(* IEC 61131-3 sources: volt/packages/volt-lsp-iec/test-corpus/lenze-mid/Device/Plc Logic/Application/A55_VarLists, 21 files *)

(* ---- Bugs.gvl ---- *)
{attribute 'qualified_only'}
{attribute 'symbol' := 'readwrite'}
VAR_GLOBAL
	checkconnection: BOOL;
	reportConnectionAlive:BOOL;
	restart: BOOL;
END_VAR

(* ---- CTE.gvl ---- *)
{attribute 'qualified_only'}
VAR_GLOBAL CONSTANT
	//TODO
	posCigarPresentOutfeed	: INT:=88;
	ct_ArraySizeCheckRegister : INT:=150;

END_VAR

(* ---- Data_Exchange_Motion.gvl ---- *)
{attribute 'qualified_only'}
VAR_GLOBAL
Servo_VirtualMaster: sUDT_VirtualMasterComm_Drive;

Servo_MainDrive: sUDT_ServoComm_Drive;
Servo_WrappingDevice: sUDT_ServoComm_Drive;
Servo_SideCorrection: sUDT_ServoComm_Drive;

FQI_FeedforwardADS : sUDT_FQIComm_Drive;
FQI_FeedforwardATF : sUDT_FQIComm_Drive;
FQI_ElevatorATF : sUDT_FQIComm_Drive;
FQI_Fan : sUDT_FQIComm_Drive;
FQI_Bobbin : sUDT_FQIComm_Drive;
BobbinTorque: DINT;

FeedForwardWrapper : sUDT_BasicMovementComm_Drive ;
END_VAR

(* ---- db_CheckRegister.gvl ---- *)
{attribute 'qualified_only'}
{attribute 'symbol' := 'readwrite'}
VAR_GLOBAL
	//Positie		: ARRAY[0..CTE.ct_ArraySizeCheckRegister] OF cUDT_ShiftRegister_Positie;
	Positie		: ARRAY[0..CTE.ct_ArraySizeCheckRegister] OF cUDT_ShiftRegister_Positie;
	EmptyCheckRegister : cUDT_ShiftRegister_Positie;
	CheckRegisterError	: BOOL;
END_VAR

(* ---- DB_Kantcorrectie.gvl ---- *)
{attribute 'qualified_only'}
{attribute 'symbol' := 'readwrite'}
VAR_GLOBAL PERSISTENT
	CopyMeasuredToLight: BOOL;
	CopyMeasuredToDark: BOOL;
	MeasuredValue		: INT;
	MeasuredValueReal	: REAL;
	Percentage			: REAL;
	Percentage10		: INT ;
	Setpoint			: INT;
	CopiedValueReal		: REAL;
	CopiedValueInt		: INT;
	LightValue			: INT:=100;
	DarkValue			: INT:=5;
	NoWrapperValue		: INT;
	DeviationNoWrapper	: INT;
	NoWrapperPercentage	: INT;
	SpareInt_2			: INT;

END_VAR

(* ---- db_MeanValuesSideCorrectionSensor.gvl ---- *)
{attribute 'qualified_only'}
VAR_GLOBAL PERSISTENT
	MeasurementValues	: ARRAY[0..50] OF INT ;
END_VAR

(* ---- Droger_Data.gvl ---- *)
{attribute 'qualified_only'}
VAR_GLOBAL
	Cor_denumerator: INT:=1;
	Cor_numerator: INT:=1;
	Act_sync_pos: INT:=1;
	Set_sync_pos: INT:=1;
END_VAR

(* ---- HMI_Interface.gvl ---- *)
{attribute 'qualified_only'}
VAR_GLOBAL
	ScreenNumber 	: sUDT_HMI_Interface_ScreenNumber;
END_VAR

(* ---- HMI_Var.gvl ---- *)
{attribute 'qualified_only'}
{attribute 'symbol' := 'readwrite'}
VAR_GLOBAL PERSISTENT RETAIN
SpareRecipe : ARRAY[0..19] OF BYTE;
RecipeNumber : Int;
DataRecordNumber : Int;
DataRecordName : String;
DownloadStatus : Int;
ResetAlarmLogging : Bool;
ForceOutputs : Bool;
RE_ForceOutputs : Bool;
Test_Prod : Bool;
Btn_Spraying : Bool;
Btn_BunchSupply : Bool;
Btn_StopLeafCarrier : Bool;
ReleaseBrake : Bool;
ManControl_1 : Bool;
ManControl_2 : Bool;
ManControl_3 : Bool;
TrayfillerActive : Bool;
Btn_DryerOn : Bool;
Btn_Cleaning : Bool;
Btn_SetIP : Bool;
HMI_AHWF_fast_winding : Bool;
SpareBool21_7 : Bool;
Led_K_Buttons : Word;
Password : Int;
HMI_AHWF_positioningType : Bool;
HMI_AHWF_StartPos : Bool;
CMD_DateTime : Bool;
Mach1: sUDT_HMIVar_Mach1;

END_VAR

(* ---- LST_General.gvl ---- *)
//{attribute 'qualified_only'}
VAR_GLOBAL
	AlwaysOn							: BOOL :=1;
	AlwaysOff							: BOOL :=0;
	FirstCycle							: BOOL:=1;

	FF50ms								: BOOL;
	Imp100ms							: BOOL;

	FF100ms								: BOOL;
	Imp200ms							: BOOL;

	FF500ms								: BOOL;
	Imp1s								: BOOL;

	FF1s								: BOOL;

	StartUpDelayPLC						: BOOL;

END_VAR

(* ---- LST_InputsOutputs.gvl ---- *)
{attribute 'qualified_only'}
VAR_GLOBAL

	//inputs
I100_0_AirpressureOK : BOOL;
I100_1_Pushbutton_start_OP0a : BOOL;
I100_2_Pushbutton_stop_OP0a : BOOL;
I100_3_Selector_switch_auto_manual_OP0a : BOOL;
I100_4_Pushbutton_request_glue_OP0a : BOOL;
I100_5_ConfigSelectionRightMachine : BOOL;
I100_6_Greasing_system_empty : BOOL;
I100_7_Spare : BOOL;

I101_0_Wrapper_present : BOOL;
I101_1_FC_Bunch_present : BOOL;
I101_2_Cigar_present : BOOL;
I101_3_Water_level_control : BOOL;
I101_4_Level_bunch_magazine : BOOL;
I101_5_Spare : BOOL;
I101_6_Toggle_greasing_cycle : BOOL;
I101_7_Spare : BOOL;

I132_0_Thermal_guards_OK : BOOL;
I132_1_PB_Start_OP2a : BOOL;
I132_2_PB_Stop_OP2a : BOOL;
I132_3_SW_Auto_Man : BOOL;
I132_4_Spare : BOOL;
I132_5_Spare : BOOL;
I132_6_Tray_down : BOOL;
I132_7_Tray_up : BOOL;

I133_0_PROX_Dryer_closed : BOOL;
I133_1_PROX_zero_position_transport_ADS : BOOL;
I133_2_Cigar_detected_at_cross_over : BOOL;
I133_3_PROX_zero_position_transport_ATF : BOOL;
I133_4_Cigar_detected_at_inpusher : BOOL;
I133_5_Spare : BOOL;
I133_6_PROX_inpusher_retracted : BOOL;
I133_7_PROX_inpusher_at_tray : BOOL;

I136_0_PROX_Elevator_above : BOOL;
I136_1_PROX_Elevator_below : BOOL;
I136_2_PROX_pulse_counter_elevator : BOOL;
I136_3_FC_Position_tray_OK : BOOL;
I136_4_PROX_Infeed_conveyor_initial_position : BOOL;
I136_5_PROX_Infeed_conveyor_at_elevator : BOOL;
I136_6_FC_Guard_tray_from_elevator : BOOL;
I136_7_FC_Outfeed_conveyor_full : BOOL;

I137_0_Spare : BOOL;
I137_1_Spare : BOOL;
I137_2_Spare : BOOL;
I137_3_Spare : BOOL;
I137_4_Spare : BOOL;
I137_5_Spare : BOOL;
I137_6_Spare : BOOL;
I137_7_Spare : BOOL;

Q100_0_Pilot_light_Alarm_green_ : BOOL;
Q100_1_Pilot_light_Alarm_orange_ : BOOL;
Q100_2_Pilot_light_Alarm_red_ : BOOL;
Q100_3_Pilot_light_Alarm_buzzer_ : BOOL;
Q100_4_Spare : BOOL;
Q100_5_Signal_lamp_Start : BOOL;
Q100_6_Signal_lamp_Stop : BOOL;
Q100_7_Activate_greasing_system : BOOL;

Q101_0_REL_release_brake : BOOL;
Q101_1_PNV_Waterlevel_control : BOOL;
Q101_2_Enable_GluePump : BOOL;
Q101_3_Spare : BOOL;
Q101_4_Spare : BOOL;
Q101_5_Spare : BOOL;
Q101_6_Spare : BOOL;
Q101_7_Spare : BOOL;

Q132_0_SL_Start_OP2a : BOOL;
Q132_1_SL_Stop_OP2a : BOOL;
Q132_2_Enable_power_controllers : BOOL;
Q132_3_Spare : BOOL;
Q132_4_CT_Fan_dryer : BOOL;
Q132_5_Spare : BOOL;
Q132_6_PNV_Inpusher : BOOL;
Q132_7_PNV_tilting_inpusher : BOOL;

Q133_0_Spare : BOOL;
Q133_1_Spare : BOOL;
Q133_2_Spare : BOOL;
Q133_3_Spare : BOOL;
Q133_4_Spare : BOOL;
Q133_5_InfeedConv_Fwd : BOOL;
Q133_6_InfeedConv_Rev : BOOL;
Q133_7_OutfeedConv_Fwd : BOOL;

Q136_0_Spare : BOOL;
Q136_1_Spare : BOOL;
Q136_2_Spare : BOOL;
Q136_3_Spare : BOOL;
Q136_4_Spare : BOOL;
Q136_5_Spare : BOOL;
Q136_6_Spare : BOOL;
Q136_7_Spare : BOOL;

Q137_0_Spare : BOOL;
Q137_1_Spare : BOOL;
Q137_2_Spare : BOOL;
Q137_3_Spare : BOOL;
Q137_4_Spare : BOOL;
Q137_5_Spare : BOOL;
Q137_6_Spare : BOOL;
Q137_7_Spare : BOOL;

{attribute 'symbol' := 'readwrite'}
IW340_LeafCoverageSensor			: INT;
{attribute 'symbol' := 'readwrite'}
Serv_QW320 : BOOL;
{attribute 'symbol' := 'readwrite'}
Serv_QW322 : BOOL;
{attribute 'symbol' := 'readwrite'}
Serv_QW324 : BOOL;

{attribute 'symbol' := 'readwrite'}
Serv_IB100 : BYTE;
{attribute 'symbol' := 'readwrite'}
Serv_IB101 : BYTE;
{attribute 'symbol' := 'readwrite'}
Serv_IB132 : BYTE;
{attribute 'symbol' := 'readwrite'}
Serv_IB133 : BYTE;
{attribute 'symbol' := 'readwrite'}
Serv_IB136 : BYTE;
{attribute 'symbol' := 'readwrite'}
Serv_IB137 : BYTE;
{attribute 'symbol' := 'readwrite'}
Serv_QB100 : BYTE;
{attribute 'symbol' := 'readwrite'}
Serv_QB101 : BYTE;
{attribute 'symbol' := 'readwrite'}
Serv_QB132 : BYTE;
{attribute 'symbol' := 'readwrite'}
Serv_QB133 : BYTE;
{attribute 'symbol' := 'readwrite'}
Serv_QB136 : BYTE;
{attribute 'symbol' := 'readwrite'}
Serv_QB137 : BYTE;
{attribute 'symbol' := 'readwrite'}
IW342_Spare : BOOL;
IW344_Spare : BOOL;
IW346_Spare : BOOL;

{attribute 'symbol' := 'readwrite'}
SMC_B0: BYTE;
{attribute 'symbol' := 'readwrite'}
SMC_B1: BYTE;
{attribute 'symbol' := 'readwrite'}
SMC_B2: BYTE;
{attribute 'symbol' := 'readwrite'}
SMC_B3: BYTE;

END_VAR

(* ---- Mach1.gvl ---- *)
{attribute 'qualified_only'}
{attribute 'symbol' := 'readwrite'}
VAR_GLOBAL
	Genflags				: UDT_GeneralFlags;
END_VAR

(* ---- Mach1_Alarms.gvl ---- *)
{attribute 'symbol' := 'readwrite'}
VAR_GLOBAL
	Mach1_Alarms	: scAlarmsDB;
	dwErrorWord1	: DWORD;
	dwErrorWord2	: DWORD;
	dwErrorWord3	: DWORD;
	dwErrorWord4	: DWORD;
END_VAR

(* ---- Mach1_AuxData.gvl ---- *)
{attribute 'qualified_only'}
VAR_GLOBAL
	AllDriveReferencingDone : BOOL;
SetDrivesInSync : Bool;
SetDrivesInLock : Bool;
AllDrivesInLock : Bool;
StartpulseDryer : Bool;
SetBuzzer : Bool;
MemContinuousGluePumping : Bool;
MemStopLeafCarrier : Bool;
MemStopCleaning : Bool;
DelayAfterDoorsActuallyClosed : Bool;
PhotocellBunchHasBeenOff : BOOL;
PhotocellCigarHasBeenOff : BOOL;
ScreenForOperatorSettingsActivated : Bool;
GlueWeighingCycleStarted : Bool;
NumberOfMutingCyclesReached : Bool;
MemLowerSpeedBecauseOfNoWrapper : Bool;
MemWrapperPresentForLeafCarrier : Bool;
MemWrapperPassedUnderTheSensor : Bool;
MemWrapperDetected_ResetLimitedSpeed : Bool;
BlockBunchInfeed : Bool;
MainDriveHomed : Bool;
RollingDeviceHomed : Bool;
DTA_Homed : Bool;
AllDrivesHomed : Bool;
CurrentCycleHasOutfeedError : Bool;
PreviousCycleHasOutfeedError : Bool;
MemCigarAtCrossOver : Bool;
ADS_StopOnZeroPulse : BOOL;
{attribute 'symbol' := 'readwrite'}
TorqueCalibrationValue : DInt;
TrayfillerActive : BOOL;
CounterHighSpeedATF_ADS: INT;
{attribute 'symbol' := 'readwrite'}
MIDS_Active : BOOL;
{attribute 'symbol' := 'readwrite'}
VelWrapperTransp : DINT;
{attribute 'symbol' := 'readwrite'}
EnableGlueSprayCalibration: BOOL:=FALSE;

{attribute 'symbol' := 'readwrite'}
EnableManualHomeSetting: BOOL:=FALSE;

IEC_TIMERS: cUDT_MachAuxData_Timers;
Edge: cUDT_MachAuxData_Edge;
COUNTERS: cUDT_MachAuxData_Counters;
ShiftRegister: cUDT_MachAuxData_Shiftregister;
CamControls : cUDT_MachAuxData_CamControls;

END_VAR

(* ---- Mach1_Data.gvl ---- *)
{attribute 'qualified_only'}
{attribute 'symbol' := 'readwrite'}
VAR_GLOBAL PERSISTENT RETAIN
MachineName : STRING;

AutoSpeed					: INT:=20;
ManualSpeed					: INT:=10;
CamControls					: cUDT_MachData_CamControls;
Timers						: cUDT_MachData_Timers;
Drives						: cUDT_MachData_Drives;
Counters					: cUDT_MachData_Counters;
Settings					: cUDT_MachData_Settings;
Dryer						: cUDT_MachData_Dryer;
TrayFiller					: cUDT_MachData_Trayfiller;

END_VAR

(* ---- Mach1_Safety.gvl ---- *)
{attribute 'qualified_only'}
{attribute 'symbol' := 'readwrite'}
VAR_GLOBAL
	Control	:	udtSafety_Control;
	Status :	udtSafety_Status;
END_VAR

(* ---- PersistentVars.gvl ---- *)
{attribute 'qualified_only'}
VAR_GLOBAL PERSISTENT RETAIN
// Generated instance path of persistent variable
	Mach1_MIDS.Mach1_Drives_DB.ServoMainDrive.STATE_Prehoming: BOOL;
	// Generated instance path of persistent variable
	Mach1_MIDS.Mach1_Drives_DB.ServoWrappingDevice.STATE_Prehoming: BOOL;
	// Generated instance path of persistent variable
	Mach1_MIDS.Mach1_Drives_DB.ServoSideCorrection.STATE_Prehoming: BOOL;
	// Generated instance path of persistent variable
	Mach1_MIDS.Mach1_Drives_DB.ServoMainDrive.STATE_HomePosNOK: BOOL;
	// Generated instance path of persistent variable
	Mach1_MIDS.Mach1_Drives_DB.ServoWrappingDevice.STATE_HomePosNOK: BOOL;
	// Generated instance path of persistent variable
	Mach1_MIDS.Mach1_Drives_DB.ServoSideCorrection.STATE_HomePosNOK: BOOL;
	// Generated instance path of persistent variable
	Mach1_MIDS.Mach1_Drives_DB.ServoMainDrive.STATE_HomePOSOK: BOOL;
	// Generated instance path of persistent variable
	Mach1_MIDS.Mach1_Drives_DB.ServoWrappingDevice.STATE_HomePOSOK: BOOL;
	// Generated instance path of persistent variable
	Mach1_MIDS.Mach1_Drives_DB.ServoSideCorrection.STATE_HomePOSOK: BOOL;
	// Generated instance path of persistent variable
	Mach1_MIDS.Mach1_Drives_DB.ServoMainDrive.STATE_WaitingForEnable: BOOL;
	// Generated instance path of persistent variable
	Mach1_MIDS.Mach1_Drives_DB.ServoWrappingDevice.STATE_WaitingForEnable: BOOL;
	// Generated instance path of persistent variable
	Mach1_MIDS.Mach1_Drives_DB.ServoSideCorrection.STATE_WaitingForEnable: BOOL;
	// Generated instance path of persistent variable
	Mach1_MIDS.Mach1_Drives_DB.ServoMainDrive.STATE_Synchronising: BOOL;
	// Generated instance path of persistent variable
	Mach1_MIDS.Mach1_Drives_DB.ServoWrappingDevice.STATE_Synchronising: BOOL;
	// Generated instance path of persistent variable
	Mach1_MIDS.Mach1_Drives_DB.ServoSideCorrection.STATE_Synchronising: BOOL;
	// Generated instance path of persistent variable

	// Generated instance path of persistent variable
	Mach1_MIDS.IDB_Dryer.stReFeedForward: R_TRIG;
	// Generated instance path of persistent variable
	Mach1_MIDS.IDB_Dryer.TMR_IntervalTimerEmptying: TON;
	// Generated instance path of persistent variable
	Mach1_MIDS.IDB_Dryer.stFaultDryerOpened: sr;
	// Generated instance path of persistent variable
	Mach1_MIDS.IDB_Dryer.stReStopFeedForward: R_TRIG;
	// Generated instance path of persistent variable
	Mach1_MIDS.IDB_Dryer.TMR_HeaterTimeOut: TON;
	// Generated instance path of persistent variable
	AHWF.IDB_WSM.stRestposition: BOOL;
	// Generated instance path of persistent variable
	AHWF.IDB_WSM.stSupplyWrapper: BOOL;
	// Generated instance path of persistent variable
	AHWF.IDB_WSM.stWrapperPresent: BOOL;
	// Generated instance path of persistent variable
	AHWF.IDB_WSM.stNoWrapper: BOOL;
	// Generated instance path of persistent variable
	AHWF.IDB_WSM.stPhotocellWrapperFault: BOOL;
	// Generated instance path of persistent variable
	AHWF.IDB_WSM.stFeedForward: BOOL;
	// Generated instance path of persistent variable
	Mach1_Data.AutoSpeed: INT;
	// Generated instance path of persistent variable
	Mach1_Data.ManualSpeed: INT;
	// Generated instance path of persistent variable
	Mach1_Data.CamControls: cUDT_MachData_CamControls;
	// Generated instance path of persistent variable
	Mach1_Data.Timers: cUDT_MachData_Timers;
	// Generated instance path of persistent variable
	Mach1_Data.Drives: cUDT_MachData_Drives;
	// Generated instance path of persistent variable
	Mach1_Data.Counters: cUDT_MachData_Counters;
	// Generated instance path of persistent variable
	Mach1_Data.Settings: cUDT_MachData_Settings;
	// Generated instance path of persistent variable
	Mach1_Data.Dryer: cUDT_MachData_Dryer;
	// Generated instance path of persistent variable
	Mach1_Data.TrayFiller: cUDT_MachData_Trayfiller;
	// Generated instance path of persistent variable
	db_MeanValuesSideCorrectionSensor.MeasurementValues: ARRAY [0..50] OF INT;
	// Generated instance path of persistent variable
	DB_Kantcorrectie.MeasuredValue: INT;
	// Generated instance path of persistent variable
	DB_Kantcorrectie.MeasuredValueReal: REAL;
	// Generated instance path of persistent variable
	DB_Kantcorrectie.Percentage: REAL;
	// Generated instance path of persistent variable
	DB_Kantcorrectie.Percentage10: INT;
	// Generated instance path of persistent variable
	DB_Kantcorrectie.Setpoint: INT;
	// Generated instance path of persistent variable
	DB_Kantcorrectie.CopiedValueReal: REAL;
	// Generated instance path of persistent variable
	DB_Kantcorrectie.CopiedValueInt: INT;
	// Generated instance path of persistent variable
	DB_Kantcorrectie.LightValue: INT;
	// Generated instance path of persistent variable
	DB_Kantcorrectie.DarkValue: INT;
	// Generated instance path of persistent variable
	DB_Kantcorrectie.NoWrapperValue: INT;
	// Generated instance path of persistent variable
	DB_Kantcorrectie.DeviationNoWrapper: INT;
	// Generated instance path of persistent variable
	DB_Kantcorrectie.NoWrapperPercentage: INT;
	// Generated instance path of persistent variable
	DB_Kantcorrectie.SpareInt_2: INT;

	//manual added values
	//AxisPosMaindrive: SMC3_PersistPosition_Data;
	//AxisPosSidecorrection: SMC3_PersistPosition_Data;
	//AxisPosWrapper: SMC3_PersistPosition_Data;

	// Generated instance path of persistent variable
	Mach1_Data.MachineName: STRING;
	// Generated instance path of persistent variable
	Mach1_MotionControl.VirtualMaster_0.lrRetainPosition: LREAL;
	// Generated instance path of persistent variable
	DB_Kantcorrectie.CopyMeasuredToLight: BOOL;
	// Generated instance path of persistent variable
	DB_Kantcorrectie.CopyMeasuredToDark: BOOL;
	// Generated instance path of persistent variable
	HMI_Var.SpareRecipe: ARRAY [0..19] OF BYTE;
	// Generated instance path of persistent variable
	HMI_Var.RecipeNumber: INT;
	// Generated instance path of persistent variable
	HMI_Var.DataRecordNumber: INT;
	// Generated instance path of persistent variable
	HMI_Var.DataRecordName: STRING;
	// Generated instance path of persistent variable
	HMI_Var.DownloadStatus: INT;
	// Generated instance path of persistent variable
	HMI_Var.ResetAlarmLogging: BOOL;
	// Generated instance path of persistent variable
	HMI_Var.ForceOutputs: BOOL;
	// Generated instance path of persistent variable
	HMI_Var.RE_ForceOutputs: BOOL;
	// Generated instance path of persistent variable
	HMI_Var.Test_Prod: BOOL;
	// Generated instance path of persistent variable
	HMI_Var.Btn_Spraying: BOOL;
	// Generated instance path of persistent variable
	HMI_Var.Btn_BunchSupply: BOOL;
	// Generated instance path of persistent variable
	HMI_Var.Btn_StopLeafCarrier: BOOL;
	// Generated instance path of persistent variable
	HMI_Var.ReleaseBrake: BOOL;
	// Generated instance path of persistent variable
	HMI_Var.ManControl_1: BOOL;
	// Generated instance path of persistent variable
	HMI_Var.ManControl_2: BOOL;
	// Generated instance path of persistent variable
	HMI_Var.ManControl_3: BOOL;
	// Generated instance path of persistent variable
	HMI_Var.TrayfillerActive: BOOL;
	// Generated instance path of persistent variable
	HMI_Var.Btn_DryerOn: BOOL;
	// Generated instance path of persistent variable
	HMI_Var.Btn_Cleaning: BOOL;
	// Generated instance path of persistent variable
	HMI_Var.Btn_SetIP: BOOL;
	// Generated instance path of persistent variable
	HMI_Var.HMI_AHWF_fast_winding: BOOL;
	// Generated instance path of persistent variable
	HMI_Var.SpareBool21_7: BOOL;
	// Generated instance path of persistent variable
	HMI_Var.Led_K_Buttons: WORD;
	// Generated instance path of persistent variable
	HMI_Var.Password: INT;
	// Generated instance path of persistent variable
	HMI_Var.HMI_AHWF_positioningType: BOOL;
	// Generated instance path of persistent variable
	HMI_Var.HMI_AHWF_StartPos: BOOL;
	// Generated instance path of persistent variable
	HMI_Var.CMD_DateTime: BOOL;
	// Generated instance path of persistent variable
	HMI_Var.Mach1: sUDT_HMIVar_Mach1;
	// Generated instance path of persistent variable
	VersionInfo_DB.PLC_version: STRING := 'ghjhggj';
	// Generated instance path of persistent variable
	VersionInfo_DB.PLC_Version_Date: STRING := 'ghjhggj';
	// Generated instance path of persistent variable
	MM_PD.scDowntime: L_OEEA_Lib.scDowntime;
	// Generated instance path of persistent variable
	MM_PD.scPDinternal: L_OEEA_Lib.scInternalVar;
	// Generated instance path of persistent variable
	MM_PD.scPDinternalDowntime: L_OEEA_Lib.scInternalDownVar;
	// Generated instance path of persistent variable
	MM_PD.scPDProductionData: L_OEEA_Lib.scInternalProductionData;
	// Generated instance path of persistent variable
	MM_PD.scPDShiftDayIndex: L_OEEA_Lib.scPDShiftData;
	// Generated instance path of persistent variable
	MM_PD.scShiftHistory: L_OEEA_Lib.scVisuShiftHistory_base;
	// Generated instance path of persistent variable
	MM_PD.scShiftDowntimeHistory: ARRAY [1..3] OF L_OEEA_Lib.scDowntime_base;
	// Generated instance path of persistent variable
	MM_PD.scOEE_VisuPD: L_OEEA_Lib.scOEE_VisuPD := STRUCT(ascVisu_OUT_ShiftTargets := [STRUCT(rOEETarget := 90.0, rOEELowerLimit := 75.0, rOEECrucial := 65.0), STRUCT(rOEETarget := 90.0, rOEELowerLimit := 75.0, rOEECrucial := 65.0), STRUCT(rOEETarget := 90.0, rOEELowerLimit := 75.0, rOEECrucial := 65.0)]);
	// Generated instance path of persistent variable
	MM_PD.scSelectedProductRecipeHMI: L_OEEA_Lib.scProduct_base;
	// Generated instance path of persistent variable
	MM_PD.sActiveProductRecipe: STRING;
	// Generated instance path of persistent variable
	MM_PD.scActiveProductRecipe: L_OEEA_Lib.scProduct_base := STRUCT(rTechnicalCycleTime := REAL#1.5, rProductTarget := 15480.0, diTypeID := DINT#1, sTypeName := 'Sigar', iUnitProductID := INT#1, sUnitProduct := 'Sigars', iUnitSpeedID := INT#1, sUnitSpeed := 'Sigars/min.', rChangeOverTime := 60.0);
	// Generated instance path of persistent variable
	MM_PD.ascDaySchedules: ARRAY [1..L_OEEA_lib.uiDaySchedule] OF L_OEEA_Lib.scDaySchedule := [7(STRUCT(iNumberofShifts := UINT_TO_INT(L_OEEA_Lib.uiNoOfShifts), iNumberofBreaks := UINT_TO_INT(L_OEEA_lib.uiNoOfBreaks), ascShiftSchedule := [STRUCT(sShiftName := 'Morning', uiStartHour := UINT#6, uiStartMinute := UINT#30, uiEndHour := UINT#14, uiEndMinute := UINT#30, uiShiftNo := UINT#1, xActive := TRUE), STRUCT(sShiftName := 'Afternoon', uiStartHour := UINT#14, uiStartMinute := UINT#30, uiEndHour := UINT#22, uiEndMinute := UINT#30, uiShiftNo := UINT#2, xActive := TRUE), STRUCT(sShiftName := 'Night', uiStartHour := UINT#22, uiStartMinute := UINT#30, uiEndHour := UINT#6, uiEndMinute := UINT#30, uiShiftNo := UINT#3, xActive := TRUE)], ascSBreakSchedule := [STRUCT(sBreakName := 'Breakfast', uiStartHour := UINT#9, uiStartMinute := UINT#0, uiEndHour := UINT#9, uiEndMinute := UINT#10, uiShiftNo := UINT#1, xActive := TRUE), STRUCT(sBreakName := 'Lunch', uiStartHour := UINT#11, uiStartMinute := UINT#0, uiEndHour := UINT#11, uiEndMinute := UINT#30, uiShiftNo := UINT#1, xActive := TRUE), STRUCT(sBreakName := 'Tea Break', uiStartHour := UINT#13, uiStartMinute := UINT#0, uiEndHour := UINT#13, uiEndMinute := UINT#10, uiShiftNo := UINT#1, xActive := TRUE), STRUCT(sBreakName := 'Tea Break 1', uiStartHour := UINT#16, uiStartMinute := UINT#0, uiEndHour := UINT#16, uiEndMinute := UINT#10, uiShiftNo := UINT#2, xActive := TRUE), STRUCT(sBreakName := 'Dinner', uiStartHour := UINT#18, uiStartMinute := UINT#45, uiEndHour := UINT#19, uiEndMinute := UINT#15, uiShiftNo := UINT#2, xActive := TRUE), STRUCT(sBreakName := 'Tea Break 2', uiStartHour := UINT#20, uiStartMinute := UINT#45, uiEndHour := UINT#20, uiEndMinute := UINT#55, uiShiftNo := UINT#2, xActive := TRUE), STRUCT(sBreakName := 'Tea Break 1', uiStartHour := UINT#23, uiStartMinute := UINT#30, uiEndHour := UINT#23, uiEndMinute := UINT#40, uiShiftNo := UINT#3, xActive := TRUE), STRUCT(sBreakName := 'Dinner', uiStartHour := UINT#1, uiStartMinute := UINT#45, uiEndHour := UINT#2, uiEndMinute := UINT#12, uiShiftNo := UINT#3, xActive := TRUE), STRUCT(sBreakName := 'Tea Break 2', uiStartHour := UINT#4, uiStartMinute := UINT#30, uiEndHour := UINT#4, uiEndMinute := UINT#40, uiShiftNo := UINT#3, xActive := TRUE)]))];
	// Generated instance path of persistent variable
	MM_PD.lrCountOK: ARRAY [1..L_OEEA_Lib.uiNoOfPartCounter] OF LREAL;
	// Generated instance path of persistent variable
	MM_PD.lrCountNOK: ARRAY [1..L_OEEA_Lib.uiNoOfPartCounter] OF LREAL;
END_VAR
%CLASS PERSISTENT

(* ---- PneumValveTerminalSMC.gvl ---- *)
{attribute 'qualified_only'}
{attribute 'symbol' := 'readwrite'}
VAR_GLOBAL
	Pos1A: BOOL;
	Pos1B: BOOL;

	Pos2A: BOOL;
	Pos2B: BOOL;
	Pos3A: BOOL;
	Pos3B: BOOL;
	Pos4A: BOOL;
	Pos4B: BOOL;
	Pos5A: BOOL;
	Pos5B: BOOL;
	Pos6A: BOOL;
	Pos6B: BOOL;

	Pos7A: BOOL;
	Pos7B: BOOL;
	Pos8A: BOOL;
	Pos8B: BOOL;
	Pos9A: BOOL;
	Pos9B: BOOL;

	Pos10A: BOOL;
	Pos10B: BOOL;
	Pos11A: BOOL;
	Pos11B: BOOL;
	Pos12A: BOOL;
	Pos12B: BOOL;

	Serv_QB202: BYTE;
	Serv_QB203: BYTE;
	Serv_QB204: BYTE;

END_VAR

(* ---- TODO.gvl ---- *)
{attribute 'qualified_only'}
VAR_GLOBAL
	//Mach1_Stop1: BOOL;
	//Mach1_Stop2: BOOL;
	//Mach1_Stop3: BOOL;
	CounterCigarAtEnd: BOOL;
	TODO_bool: BOOL;
	//stopdrive_test1:BOOL;
	//stopdrive_test2:BOOL;
	//stopdrive_test3:BOOL;
	//stopdrive_test4:BOOL;
	//stopdrive_test5:BOOL;
	//stopdrive_test6:BOOL;
	//stopdrive_test7:BOOL;
	//stopdrive_test8:BOOL;
	//stopdrive_test9:BOOL;

END_VAR

(* ---- Trayfiller_Data.gvl ---- *)
{attribute 'qualified_only'}
VAR_GLOBAL
	Alarms	:	cUDT_Trayfiller_Data_Alarms;
	commInterface	: cUDT_Trafiller_Data_Interface;

END_VAR

(* ---- VersionInfo_DB.gvl ---- *)
{attribute 'qualified_only'}
{attribute 'symbol' := 'readwrite'}
VAR_GLOBAL PERSISTENT RETAIN
	PLC_version: STRING:='ghjhggj';
	PLC_Version_Date: STRING:='ghjhggj';

END_VAR
